KUKA KRL program: wkz3_ab.src, wkz3_ab.dat

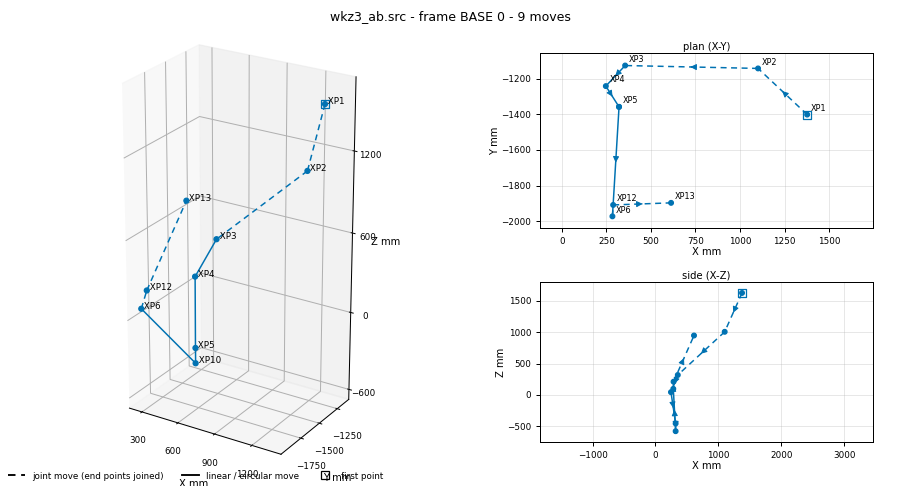
[picture p0: tool path of wkz3_ab.src in frame BASE 0, 9 of 9 moves have a stored position in this frame; points joined in program order, loops and branches not executed]
--- wkz3_ab.src ---
&ACCESS RVO2
&REL 125
&COMMENT DEP_GRIPPER_ACCELO
&PARAM DISKPATH = KRC:\R1\Program\WKZ
DEF WKZ3_AB ( )
;FOLD INI
  ;FOLD BASISTECH INI
    GLOBAL INTERRUPT DECL 3 WHEN $STOPMESS==TRUE DO IR_STOPM ( )
    INTERRUPT ON 3
    BAS (#INITMOV,0 )
  ;ENDFOLD (BASISTECH INI)
  ;FOLD USER INI
    ;Make your modifications here
  ;ENDFOLD (USER INI)
;ENDFOLD (INI)
; Caracterização dos meios de produção:
; Versão Atual:
; 04/05/2013 12:00 Name: P13.090-R6 CHANGES: Deposita Garra
; Accelo

chk_W3_wechs_ok ( )  ; VERIFICAÇÃO DE FERRAMENTA: GRIPPER ACELLO

;FOLD SET GRP 5 State=CLO GDAT3;%{PE}%R 8.2.4,%MKUKATPGRP,%CGRP,%VGRP,%P 2:5, 4:1, 5:#NO, 6:GDAT3, 8:1, 10:0
H50(GRP,5,1,GGDAT3)
;ENDFOLD
chk_w3_grp5_opn ()

;FOLD SET GRP 6 State=CLO GDAT4;%{PE}%R 8.2.4,%MKUKATPGRP,%CGRP,%VGRP,%P 2:6, 4:1, 5:#NO, 6:GDAT4, 8:1, 10:0
H50(GRP,6,1,GGDAT4)
;ENDFOLD
chk_w3_grp6_opn ()

;FOLD PTP P1 Vel=100 % PDAT1 Tool[3]:Gripper Parabrisa Accelo Base[0];%{PE}%R 8.2.24,%MKUKATPBASIS,%CMOVE,%VPTP,%P 1:PTP, 2:P1, 3:, 5:100, 7:PDAT1
$BWDSTART=FALSE
PDAT_ACT=PPDAT1
FDAT_ACT=FP1
BAS(#PTP_PARAMS,100)
PTP XP1
;ENDFOLD
;FOLD PTP P2 CONT Vel=100 % PDAT2 Tool[3]:Gripper Parabrisa Accelo Base[0];%{PE}%R 8.2.24,%MKUKATPBASIS,%CMOVE,%VPTP,%P 1:PTP, 2:P2, 3:C_PTP, 5:100, 7:PDAT2
$BWDSTART=FALSE
PDAT_ACT=PPDAT2
FDAT_ACT=FP2
BAS(#PTP_PARAMS,100)
PTP XP2 C_PTP
;ENDFOLD

;FOLD WAIT FOR ( NOT IN 177 'DEPOSITO 3 OCUPADO' );%{PE}%R 8.2.24,%MKUKATPBASIS,%CEXT_WAIT_FOR,%VEXT_WAIT_FOR,%P 2:, 4:NOT, 5:$IN, 6:177, 7:DEPOSITO 3 OCUPADO, 9:
WAIT FOR  (  NOT $IN[177] )
;ENDFOLD
;FOLD WAIT FOR ( IN 219 'PLACA DE SUPORTE FUNDIDA' );%{PE}%R 8.2.24,%MKUKATPBASIS,%CEXT_WAIT_FOR,%VEXT_WAIT_FOR,%P 2:, 4:, 5:$IN, 6:219, 7:PLACA DE SUPORTE FUNDIDA, 9:
WAIT FOR  ( $IN[219] )
;ENDFOLD
;FOLD PULSE 183 'Proteção da pinca 3 abrir' State=TRUE Time=0.3 sec;%{PE}%R 8.2.24,%MKUKATPBASIS,%COUT,%VPULSE,%P 2:183, 3:Proteção da pinca 3 abrir, 5:TRUE, 6:, 8:0.3
PULSE($OUT[183], TRUE,0.3)
;ENDFOLD
;FOLD WAIT FOR ( IN 181 'PROTECAO DE PINCA ABERTA' );%{PE}%R 8.2.24,%MKUKATPBASIS,%CEXT_WAIT_FOR,%VEXT_WAIT_FOR,%P 2:, 4:, 5:$IN, 6:181, 7:PROTECAO DE PINCA ABERTA, 9:
WAIT FOR  ( $IN[181] )
;ENDFOLD
;FOLD WAIT FOR ( NOT IN 182 'PROTECAO DE PINCA FECHADA' );%{PE}%R 8.2.24,%MKUKATPBASIS,%CEXT_WAIT_FOR,%VEXT_WAIT_FOR,%P 2:, 4:NOT, 5:$IN, 6:182, 7:PROTECAO DE PINCA FECHADA, 9:
WAIT FOR  (  NOT $IN[182] )
;ENDFOLD

;FOLD PTP P3 CONT Vel=100 % PDAT3 Tool[3]:Gripper Parabrisa Accelo Base[0];%{PE}%R 8.2.24,%MKUKATPBASIS,%CMOVE,%VPTP,%P 1:PTP, 2:P3, 3:C_PTP, 5:100, 7:PDAT3
$BWDSTART=FALSE
PDAT_ACT=PPDAT3
FDAT_ACT=FP3
BAS(#PTP_PARAMS,100)
PTP XP3 C_PTP
;ENDFOLD
;FOLD LIN P4 CONT Vel=0.5 m/s CPDAT1 Tool[3]:Gripper Parabrisa Accelo Base[0];%{PE}%R 8.2.24,%MKUKATPBASIS,%CMOVE,%VLIN,%P 1:LIN, 2:P4, 3:C_DIS, 5:0.5, 7:CPDAT1
$BWDSTART=FALSE
LDAT_ACT=LCPDAT1
FDAT_ACT=FP4
BAS(#CP_PARAMS,0.5)
LIN XP4 C_DIS
;ENDFOLD
;FOLD LIN P5 Vel=0.5 m/s CPDAT2 Tool[3]:Gripper Parabrisa Accelo Base[0];%{PE}%R 8.2.24,%MKUKATPBASIS,%CMOVE,%VLIN,%P 1:LIN, 2:P5, 3:, 5:0.5, 7:CPDAT2
$BWDSTART=FALSE
LDAT_ACT=LCPDAT2
FDAT_ACT=FP5
BAS(#CP_PARAMS,0.5)
LIN XP5
;ENDFOLD

;FOLD ; Ponto de deposito GARRA ACCELO;%{PE}%R 8.2.24,%MKUKATPBASIS,%CCOMMENT,%VNORMAL,%P 2:Ponto  de deposito  GARRA ACCELO
;ENDFOLD
;FOLD LIN P10 Vel=0.1 m/s CPDAT5 Tool[3]:Gripper Parabrisa Accelo Base[0];%{PE}%R 8.2.24,%MKUKATPBASIS,%CMOVE,%VLIN,%P 1:LIN, 2:P10, 3:, 5:0.1, 7:CPDAT5
$BWDSTART=FALSE
LDAT_ACT=LCPDAT5
FDAT_ACT=FP10
BAS(#CP_PARAMS,0.1)
LIN XP10
;ENDFOLD

;FOLD WAIT FOR ( IN 177 'DEPOSITO 3 OCUPADO' );%{PE}%R 8.2.24,%MKUKATPBASIS,%CEXT_WAIT_FOR,%VEXT_WAIT_FOR,%P 2:, 4:, 5:$IN, 6:177, 7:DEPOSITO 3 OCUPADO, 9:
WAIT FOR  ( $IN[177] )
;ENDFOLD

;FOLD OUT 223 'DESBLOQUEIA MPS' State=TRUE ;%{PE}%R 8.2.24,%MKUKATPBASIS,%COUT,%VOUTX,%P 2:223, 3:DESBLOQUEIA MPS, 5:TRUE, 6:
$OUT[223]=TRUE
;ENDFOLD
;FOLD OUT 224 'BLOQUEIA MPS' State=FALSE ;%{PE}%R 8.2.24,%MKUKATPBASIS,%COUT,%VOUTX,%P 2:224, 3:BLOQUEIA MPS, 5:FALSE, 6:
$OUT[224]=FALSE
;ENDFOLD

;FOLD WAIT FOR ( IN 217 'MPS DESTRAVADO' );%{PE}%R 8.2.24,%MKUKATPBASIS,%CEXT_WAIT_FOR,%VEXT_WAIT_FOR,%P 2:, 4:, 5:$IN, 6:217, 7:MPS DESTRAVADO, 9:
WAIT FOR  ( $IN[217] )
;ENDFOLD
;FOLD WAIT FOR ( NOT IN 221 'MPS TRAVADO' );%{PE}%R 8.2.24,%MKUKATPBASIS,%CEXT_WAIT_FOR,%VEXT_WAIT_FOR,%P 2:, 4:NOT, 5:$IN, 6:221, 7:MPS TRAVADO, 9:
WAIT FOR  (  NOT $IN[221] )
;ENDFOLD

;FOLD IBUS OFF;%{PE}%R 8.2.24,%MKUKATPBASIS,%CIBUS,%VMAP,%P 2:#OFF, 3:1
$IBUS_OFF=$IBUS_ON
$IBUS_ON=0
;ENDFOLD
;FOLD WAIT Time=1.5 sec;%{PE}%R 8.2.24,%MKUKATPBASIS,%CWAIT,%VWAIT,%P 3:1.5
WAIT SEC 1.5
;ENDFOLD

;FOLD LIN P6 CONT Vel=0.5 m/s CPDAT3 Tool[8]:Tool Changer Base[0];%{PE}%R 8.2.24,%MKUKATPBASIS,%CMOVE,%VLIN,%P 1:LIN, 2:P6, 3:C_DIS, 5:0.5, 7:CPDAT3
$BWDSTART=FALSE
LDAT_ACT=LCPDAT3
FDAT_ACT=FP6
BAS(#CP_PARAMS,0.5)
LIN XP6 C_DIS
;ENDFOLD

;FOLD WAIT FOR ( NOT IN 219 'PLACA DE SUPORTE FUNDIDA' );%{PE}%R 8.2.24,%MKUKATPBASIS,%CEXT_WAIT_FOR,%VEXT_WAIT_FOR,%P 2:, 4:NOT, 5:$IN, 6:219, 7:PLACA DE SUPORTE FUNDIDA, 9:
WAIT FOR  (  NOT $IN[219] )
;ENDFOLD
;FOLD WAIT FOR ( IN 177 'DEPOSITO 3 OCUPADO' );%{PE}%R 8.2.24,%MKUKATPBASIS,%CEXT_WAIT_FOR,%VEXT_WAIT_FOR,%P 2:, 4:, 5:$IN, 6:177, 7:DEPOSITO 3 OCUPADO, 9:
WAIT FOR  ( $IN[177] )
;ENDFOLD

;FOLD OUT 223 'DESBLOQUEIA MPS' State=FALSE ;%{PE}%R 8.2.24,%MKUKATPBASIS,%COUT,%VOUTX,%P 2:223, 3:DESBLOQUEIA MPS, 5:FALSE, 6:
$OUT[223]=FALSE
;ENDFOLD
;FOLD OUT 224 'BLOQUEIA MPS' State=TRUE ;%{PE}%R 8.2.24,%MKUKATPBASIS,%COUT,%VOUTX,%P 2:224, 3:BLOQUEIA MPS, 5:TRUE, 6:
$OUT[224]=TRUE
;ENDFOLD

;FOLD PTP P12 CONT Vel=100 % PDAT7 Tool[8]:Tool Changer Base[0];%{PE}%R 8.2.24,%MKUKATPBASIS,%CMOVE,%VPTP,%P 1:PTP, 2:P12, 3:C_PTP, 5:100, 7:PDAT7
$BWDSTART=FALSE
PDAT_ACT=PPDAT7
FDAT_ACT=FP12
BAS(#PTP_PARAMS,100)
PTP XP12 C_PTP
;ENDFOLD
;FOLD PTP P13 Vel=100 % PDAT8 Tool[8]:Tool Changer Base[0];%{PE}%R 8.2.24,%MKUKATPBASIS,%CMOVE,%VPTP,%P 1:PTP, 2:P13, 3:, 5:100, 7:PDAT8
$BWDSTART=FALSE
PDAT_ACT=PPDAT8
FDAT_ACT=FP13
BAS(#PTP_PARAMS,100)
PTP XP13
;ENDFOLD

;FOLD PULSE 184 'Proteção da pinca 3 fechar' State=TRUE Time=0.3 sec;%{PE}%R 8.2.24,%MKUKATPBASIS,%COUT,%VPULSE,%P 2:184, 3:Proteção da pinca 3 fechar, 5:TRUE, 6:, 8:0.3
PULSE($OUT[184], TRUE,0.3)
;ENDFOLD

END

--- wkz3_ab.dat ---
&ACCESS RVO2
&REL 125
&COMMENT DEP_GRIPPER_ACCELO
&PARAM DISKPATH = KRC:\R1\Program\WKZ
DEFDAT  wkz3_ab
;FOLD EXTERNAL DECLARATIONS;%{PE}%MKUKATPBASIS,%CEXT,%VCOMMON,%P
;FOLD BASISTECH EXT;%{PE}%MKUKATPBASIS,%CEXT,%VEXT,%P
EXT  BAS (BAS_COMMAND  :IN,REAL  :IN )
DECL INT SUCCESS
;ENDFOLD (BASISTECH EXT)
;FOLD USER EXT;%{E}%MKUKATPUSER,%CEXT,%VEXT,%P
;Make your modifications here
;ENDFOLD (USER EXT)
;ENDFOLD (EXTERNAL DECLARATIONS)

;# ============ START PATH : wkz3_ab =============
DECL FDAT Fnew_wkz3_ab_p37={TOOL_NO 3,BASE_NO 0,IPO_FRAME #BASE,POINT2[] " "}
DECL PDAT PP_OLP1={VEL 100.0,ACC 100.0,APO_DIST 0.0}
DECL E6POS Xnew_wkz3_ab_p37={X 1376.823,Y -1401.60999,Z 1623.00403,A -28.9843006,B -54.9752007,C 168.858994,S 2,T 2}
DECL FDAT Fnew_wkz3_ab_p14={TOOL_NO 3,BASE_NO 0,IPO_FRAME #BASE,POINT2[] " "}
DECL PDAT PP_OLP2={VEL 100.0,ACC 100.0,APO_DIST 0.0}
DECL E6POS Xnew_wkz3_ab_p14={X 1101.28003,Y -1142.50403,Z 1004.95801,A -29.1103001,B -30.0618992,C 172.812805,S 2,T 2}
DECL FDAT Fnew_wkz3_ab_p10={TOOL_NO 3,BASE_NO 0,IPO_FRAME #BASE,POINT2[] " "}
DECL PDAT PP_OLP3={VEL 100.0,ACC 100.0,APO_DIST 0.0}
DECL E6POS Xnew_wkz3_ab_p10={X 355.096985,Y -1126.22302,Z 317.803986,A -1.22749996,B 6.41580009,C -179.961899,S 2,T 2}
DECL FDAT Fnew_wkz3_ab_p25={TOOL_NO 3,BASE_NO 0,IPO_FRAME #BASE,POINT2[] " "}
DECL E6POS Xnew_wkz3_ab_p25={X 246.75,Y -1241.69702,Z 44.9099998,A -1.22609997,B 6.4144001,C -179.959,S 2,T 2}
DECL LDAT LL_OLP1={VEL 0.5,ACC 100.0,APO_DIST 10.0,APO_FAC 50.0,ORI_TYP #VAR,CIRC_TYP #BASE,JERK_FAC 50.0}
DECL FDAT Fnew_wkz3_ab_p35={TOOL_NO 3,BASE_NO 0,IPO_FRAME #BASE,POINT2[] " "}
DECL E6POS Xnew_wkz3_ab_p35={X 246.024994,Y -1298.22302,Z -267.679993,A -1.22870004,B 5.79890013,C -179.955002,S 2,T 2}
DECL LDAT LL_OLP2={VEL 0.5,ACC 100.0,APO_DIST 10.0,APO_FAC 50.0,ORI_TYP #VAR,CIRC_TYP #BASE,JERK_FAC 50.0}
DECL FDAT Fnew_wkz3_ab_p36={TOOL_NO 3,BASE_NO 0,IPO_FRAME #BASE,POINT2[] " "}
DECL E6POS Xnew_wkz3_ab_p36={X 288.816986,Y -1299.11206,Z -419.725006,A -1.23029995,B 3.31900001,C -179.957901,S 2,T 2}
DECL LDAT LL_OLP3={VEL 0.5,ACC 100.0,APO_DIST 10.0,APO_FAC 50.0,ORI_TYP #VAR,CIRC_TYP #BASE,JERK_FAC 50.0}
DECL FDAT Fnew_wkz3_ab_p11={TOOL_NO 3,BASE_NO 0,IPO_FRAME #BASE,POINT2[] " "}
DECL E6POS Xnew_wkz3_ab_p11={X 304.971985,Y -1299.68799,Z -562.179993,A -1.23179996,B 0.969399989,C -179.971603,S 2,T 2}
DECL LDAT LL_OLP4={VEL 0.5,ACC 100.0,APO_DIST 5.0,APO_FAC 50.0,ORI_TYP #VAR,CIRC_TYP #BASE,JERK_FAC 50.0}
DECL FDAT Fnew_wkz3_ab_p12={TOOL_NO 8,BASE_NO 0,IPO_FRAME #BASE,POINT2[] " "}
DECL E6POS Xnew_wkz3_ab_p12={X 279.942993,Y -2042.16003,Z -24.2310009,A 11.8758001,B 8.36009979,C 151.335297,S 2,T 2}
DECL LDAT LL_OLP5={VEL 0.25,ACC 100.0,APO_DIST 0.0,APO_FAC 0.0,ORI_TYP #VAR,CIRC_TYP #BASE,JERK_FAC 50.0}
DECL FDAT Fnew_wkz3_ab_p13={TOOL_NO 8,BASE_NO 0,IPO_FRAME #BASE,POINT2[] " "}
DECL E6POS Xnew_wkz3_ab_p13={X 280.43399,Y -2032.76697,Z -7.78399992,A 11.8755999,B 8.35999966,C 151.335297,S 2,T 2}
DECL LDAT LL_OLP6={VEL 0.25,ACC 100.0,APO_DIST 0.0,APO_FAC 0.0,ORI_TYP #VAR,CIRC_TYP #BASE,JERK_FAC 50.0}
DECL FDAT Fnew_wkz3_ab_p15={TOOL_NO 8,BASE_NO 0,IPO_FRAME #BASE,POINT2[] " "}
DECL PDAT PP_OLP4={VEL 100.0,ACC 100.0,APO_DIST 0.0}
DECL E6POS Xnew_wkz3_ab_p15={X 286.071014,Y -1944.13403,Z 149.699005,A 11.8761997,B 8.35719967,C 151.173599,S 2,T 2}
DECL FDAT Fnew_wkz3_ab_p26={TOOL_NO 8,BASE_NO 0,IPO_FRAME #BASE,POINT2[] " "}
DECL PDAT PP_OLP5={VEL 100.0,ACC 100.0,APO_DIST 0.0}
DECL E6POS Xnew_wkz3_ab_p26={X 695.919006,Y -1943.66296,Z 886.799011,A -103.576103,B -23.6098995,C -178.892593,S 2,T 2}
DECL BASIS_SUGG_T LAST_BASIS={POINT1[] "P13                     ",POINT2[] "P13                     ",CP_PARAMS[] "CPDAT5                  ",PTP_PARAMS[] "PDAT8                   ",CONT[] "C_PTP                   ",CP_VEL[] "0.5                     ",PTP_VEL[] "100                     ",SYNC_PARAMS[] "SYNCDAT                 ",SPL_NAME[] "S0                      "}
DECL E6POS XP1={X 1376.828,Y -1401.61597,Z 1623.01001,A -28.9869499,B -54.9751892,C 168.861206,S 18,T 2,E1 0.0,E2 0.0,E3 0.0,E4 0.0,E5 0.0,E6 0.0}
DECL FDAT FP1={TOOL_NO 3,BASE_NO 0,IPO_FRAME #BASE,POINT2[] " ",TQ_STATE FALSE}
DECL PDAT PPDAT1={VEL 100.0,ACC 50.0,APO_DIST 100.0,GEAR_JERK 50.0}
DECL E6POS XP2={X 1101.27502,Y -1142.5,Z 1004.94897,A -29.1102905,B -30.0612106,C 172.813202,S 18,T 2,E1 0.0,E2 0.0,E3 0.0,E4 0.0,E5 0.0,E6 0.0}
DECL FDAT FP2={TOOL_NO 3,BASE_NO 0,IPO_FRAME #BASE,POINT2[] " ",TQ_STATE FALSE}
DECL PDAT PPDAT2={VEL 100.0,ACC 100.0,APO_DIST 0.0,APO_MODE #CPTP,GEAR_JERK 50.0}
DECL E6POS XP3={X 355.136902,Y -1126.21204,Z 317.804504,A -1.22945797,B 6.41449308,C -179.961197,S 18,T 2,E1 0.0,E2 0.0,E3 0.0,E4 0.0,E5 0.0,E6 0.0}
DECL FDAT FP3={TOOL_NO 3,BASE_NO 0,IPO_FRAME #BASE,POINT2[] " ",TQ_STATE FALSE}
DECL PDAT PPDAT3={VEL 100.0,ACC 50.0,APO_DIST 0.0,APO_MODE #CPTP,GEAR_JERK 50.0}
DECL E6POS XP4={X 246.762207,Y -1241.68701,Z 44.9111595,A -1.22619605,B 6.41403008,C -179.958496,S 18,T 2,E1 0.0,E2 0.0,E3 0.0,E4 0.0,E5 0.0,E6 0.0}
DECL FDAT FP4={TOOL_NO 3,BASE_NO 0,IPO_FRAME #BASE,POINT2[] " ",TQ_STATE FALSE}
DECL LDAT LCPDAT1={VEL 2.0,ACC 100.0,APO_DIST 100.0,APO_FAC 50.0,AXIS_VEL 100.0,AXIS_ACC 100.0,ORI_TYP #VAR,CIRC_TYP #BASE,JERK_FAC 50.0,GEAR_JERK 50.0,EXAX_IGN 0}
DECL E6POS XP5={X 320.732208,Y -1358.08606,Z -453.482788,A -1.25441504,B 1.00945902,C -179.808105,S 18,T 2,E1 0.0,E2 0.0,E3 0.0,E4 0.0,E5 0.0,E6 0.0}
DECL FDAT FP5={TOOL_NO 3,BASE_NO 0,IPO_FRAME #BASE,POINT2[] " ",TQ_STATE FALSE}
DECL LDAT LCPDAT2={VEL 2.0,ACC 100.0,APO_DIST 10.0,APO_FAC 50.0,AXIS_VEL 100.0,AXIS_ACC 100.0,ORI_TYP #VAR,CIRC_TYP #BASE,JERK_FAC 50.0,GEAR_JERK 50.0,EXAX_IGN 0}
DECL E6POS XP6={X 283.769196,Y -1972.77002,Z 97.6769867,A 11.8715801,B 8.35883904,C 151.330795,S 18,T 2,E1 0.0,E2 0.0,E3 0.0,E4 0.0,E5 0.0,E6 0.0}
DECL FDAT FP6={TOOL_NO 8,BASE_NO 0,IPO_FRAME #BASE,POINT2[] " ",TQ_STATE FALSE}
DECL LDAT LCPDAT3={VEL 2.0,ACC 100.0,APO_DIST 10.0,APO_FAC 50.0,AXIS_VEL 100.0,AXIS_ACC 100.0,ORI_TYP #VAR,CIRC_TYP #BASE,JERK_FAC 50.0,GEAR_JERK 50.0,EXAX_IGN 0}
DECL E6POS XP7={X 308.408508,Y -1370.80298,Z -386.560608,A -1.70786703,B 2.86060905,C 179.407104,S 18,T 2,E1 0.0,E2 0.0,E3 0.0,E4 0.0,E5 0.0,E6 0.0}
DECL FDAT FP7={TOOL_NO 3,BASE_NO 0,IPO_FRAME #BASE,POINT2[] " ",TQ_STATE FALSE}
DECL PDAT PPDAT4={VEL 100.0,ACC 100.0,APO_DIST 100.0,APO_MODE #CPTP,GEAR_JERK 50.0}
DECL LDAT LCPDAT4={VEL 2.0,ACC 100.0,APO_DIST 100.0,APO_FAC 50.0,AXIS_VEL 100.0,AXIS_ACC 100.0,ORI_TYP #VAR,CIRC_TYP #BASE,JERK_FAC 50.0,GEAR_JERK 50.0,EXAX_IGN 0}
DECL E6POS XP8={X 279.774292,Y -2045.61304,Z -30.3410301,A 11.8758802,B 8.35905361,C 151.336807,S 18,T 2,E1 0.0,E2 0.0,E3 0.0,E4 0.0,E5 0.0,E6 0.0}
DECL FDAT FP8={TOOL_NO 8,BASE_NO 0,IPO_FRAME #BASE,POINT2[] " ",TQ_STATE FALSE}
DECL E6POS XP9={X 320.680511,Y -1358.05603,Z -453.470215,A -1.25201094,B 1.01146102,C -179.807098,S 18,T 2,E1 0.0,E2 0.0,E3 0.0,E4 0.0,E5 0.0,E6 0.0}
DECL FDAT FP9={TOOL_NO 3,BASE_NO 0,IPO_FRAME #BASE,POINT2[] " ",TQ_STATE FALSE}
DECL PDAT PPDAT5={VEL 100.0,ACC 100.0,APO_DIST 100.0,APO_MODE #CPTP,GEAR_JERK 50.0}
DECL E6POS XP10={X 320.944702,Y -1358.16895,Z -576.118225,A -1.25678003,B 1.00527,C -179.816299,S 18,T 2,E1 0.0,E2 0.0,E3 0.0,E4 0.0,E5 0.0,E6 0.0}
DECL FDAT FP10={TOOL_NO 3,BASE_NO 0,IPO_FRAME #BASE,POINT2[] " ",TQ_STATE FALSE}
DECL LDAT LCPDAT5={VEL 2.0,ACC 100.0,APO_DIST 100.0,APO_FAC 50.0,AXIS_VEL 100.0,AXIS_ACC 100.0,ORI_TYP #VAR,CIRC_TYP #BASE,JERK_FAC 50.0,GEAR_JERK 50.0,EXAX_IGN 0}
DECL E6POS XP11={X 320.944702,Y -1358.16895,Z -576.117798,A -1.25675702,B 1.00527203,C -179.816299,S 18,T 2,E1 0.0,E2 0.0,E3 0.0,E4 0.0,E5 0.0,E6 0.0}
DECL FDAT FP11={TOOL_NO 3,BASE_NO 0,IPO_FRAME #BASE,POINT2[] " ",TQ_STATE FALSE}
DECL PDAT PPDAT6={VEL 100.0,ACC 100.0,APO_DIST 100.0,GEAR_JERK 50.0}
DECL E6POS XP12={X 287.934113,Y -1908.71997,Z 211.3526,A 11.8753796,B 8.35694122,C 151.175003,S 18,T 2,E1 0.0,E2 0.0,E3 0.0,E4 0.0,E5 0.0,E6 0.0}
DECL FDAT FP12={TOOL_NO 8,BASE_NO 0,IPO_FRAME #BASE,POINT2[] " ",TQ_STATE FALSE}
DECL PDAT PPDAT7={VEL 100.0,ACC 100.0,APO_DIST 100.0,APO_MODE #CPTP,GEAR_JERK 50.0}
DECL E6POS XP13={X 612.972229,Y -1897.00806,Z 945.962891,A -103.577301,B -23.6069393,C -178.894302,S 18,T 2,E1 0.0,E2 0.0,E3 0.0,E4 0.0,E5 0.0,E6 0.0}
DECL FDAT FP13={TOOL_NO 8,BASE_NO 0,IPO_FRAME #BASE,POINT2[] " ",TQ_STATE FALSE}
DECL PDAT PPDAT8={VEL 100.0,ACC 100.0,APO_DIST 0.0,APO_MODE #CPTP,GEAR_JERK 50.0}
DECL GRP_SUGG_T LAST_GRP={NUMBER[] "6                       ",STATE[] "2                       ",PARAMS[] "GDAT2                   "}
DECL GRP_TYP GGDAT1={G_APO #NO,GRP_TIME 0.200000003,CTRL #OFF,DLY 0,DST 1}
DECL GRP_TYP GGDAT2={G_APO #NO,GRP_TIME 0.200000003,CTRL #OFF,DLY 0,DST 1}
DECL GRP_TYP GGDAT3={G_APO #NO,GRP_TIME 0.200000003,CTRL #OFF,DLY 0,DST 1}
DECL GRP_TYP GGDAT4={G_APO #NO,GRP_TIME 0.200000003,CTRL #OFF,DLY 0,DST 1}
ENDDAT
